Staubli VAL3: remSetTCPVals.pgx

program remSetTCPVals(string& sArgs[] (dimensions=1), string& sReturn[] (dimensions=1))
  local bool bOk
  local num nArg
  local num nTemp
  local trsf trTCP
begin
  // Set the values of the TCP
  //
  // Arguments are "X Y Z RX RY RZ"
  //
  logMsg("call remSetTCPVals")
  nArg=0
  trTCP={0,0,0,0,0,0}
  while nArg<6
    sArgs=toNum(sArgs,nTemp,bOk)
    if bOk
      switch nArg
        case 0
          trTCP.x=nTemp
        break
        case 1
          trTCP.y=nTemp
        break
        case 2
          trTCP.z=nTemp
        break
        case 3
          trTCP.rx=nTemp
        break
        case 4
          trTCP.ry=nTemp
        break
        case 5
          trTCP.rz=nTemp
        break
      endSwitch
      nArg=nArg+1
    else
      call remErrNum("SETTCPVALS",sArgs,sReturn)
      return
    endIf
  endWhile
  tSensorTool.trsf=trTCP
  sReturn="SETTCPVALS"
end
